FUNCTION_BLOCK EL3182
VAR
	_io : EL3xx2_Data;
	{attribute addProperty Name "WcState"}
	_wcState : WcStateInputToggle;
	{attribute addProperty Name "Info data"}
	_infoData : InfoDataAdsAoE;
END_VAR

PROPERTY IO : REFERENCE TO EL3xx2_Data
GET
IO REF= _io;
END_GET
END_PROPERTY

PROPERTY WcState : REFERENCE TO WcStateInputToggle
GET
WcState REF= _wcState;
END_GET
END_PROPERTY

END_FUNCTION_BLOCK

(* stored: Version 1.1.0.1, ProductVersion 3.1.4024.9
   POU EL3182: Id {c0f4f506-f3b2-0e0e-2f3e-20362a0cd698}, SpecialFunc None
   Property IO: Id {592f989d-bf58-0345-3694-436bcbd35910}
   Get Get: Id {d55c4051-b2a2-0c16-325e-d09b171c1592}
   Property WcState: Id {6d37f781-d261-0447-0533-d8c413580d28}
   Get Get: Id {8b7eef9f-a926-0a62-24d2-e0f8aa7ca23d} *)
